// TwinCAT 3 PLC project ADSMotion
// ProgramVersion: 3.1.4024.0
// libraries:
//   Tc2_DataExchange, * (Beckhoff Automation GmbH)
//   Tc2_MC2, * (Beckhoff Automation GmbH)
//   Tc2_Standard, * (Beckhoff Automation GmbH)
//   Tc2_System, * (Beckhoff Automation GmbH)
//   Tc3_Module, * (Beckhoff Automation GmbH)
// project tree:
//   DUTs/ ST_variables.TcDUT
//   / PlcTask.TcTTO
//   POUs/ MAIN.TcPOU
// real-time tasks:
//   TASK PlcTask: cycle T#10ms, priority 20, ADS port 350
// motion (NC):
//   TASK NC-Task 1 SAF: cycle T#10ms, priority 4, ADS port 501
//   TASK NC-Task 1 SVB: cycle T#10ms, priority 8, ADS port 511
//   AXIS Axis 1 (id 1)
//     OtherSettings: AllowMotionCmdToSlave=true
//     encoder EncType=1
//     drive DrvType=5
//       Analog: TorqueSetpointScale=10, ScaleFactorActTorque=0.1
//       TimeComp: TaskDelayCycles=1
//     controller CtrType=1
//       CtrPara: PriorControlFactor=1
//         Observer: BandWidth=20

CONFIGURATION ADSMotion
    RESOURCE PLC ON TwinCAT3
        TASK PlcTask(INTERVAL := T#10ms, PRIORITY := 20);
        PROGRAM MAIN WITH PlcTask : MAIN;
    END_RESOURCE
END_CONFIGURATION

// ---- DUTs/ST_variables.TcDUT
TYPE ST_variables :
STRUCT
	bEnable   : BOOL;
    bStop     : BOOL;
    bMoveRel  : BOOL;
    rVelocity : REAL;
    rDistance : REAL;
END_STRUCT
END_TYPE

// ---- POUs/MAIN.TcPOU
PROGRAM MAIN
VAR
	//Write BOOL and REAL
	fbADSBoolEnable		: FB_WriteBoolOnDelta;
	fbADSBoolStop 		: FB_WriteBoolOnDelta;
	fbADSBoolRelMove 	: FB_WriteBoolOnDelta;
	fbADSRealVelocity	: FB_WriteRealOnDelta;
	fbADSRealDistance	: FB_WriteRealOnDelta;
	
    //ADS Comms Watchdoog
    fbWrWd : FB_WriteWatchdog;

		
	bEnabletx 		:BOOL; //Enable Controller
	bStoptx			: BOOL;
	bMoveReltx		: BOOL;
	rVelocitytx		: REAL;
	rDistancetx		: REAL;

	
END_VAR

fbWrWd(
    bEnable       := TRUE,
    sNetId        := '10.200.228.35.1.1',
    nPort         := 851,
    sVarName      := 'MAIN.nWatchdogRx',
    tWatchdogTime := T#1S
);

fbADSBoolEnable(
	bEnable:= TRUE , 
	sNetId:= '10.200.228.35.1.1', 
	nPort:= 851 , 
	sVarName:= 'MAIN.bEnable' , 
	bSignal:= bEnabletx , 
	tCycleTime:= T#1MS , 
	bSendNow:= FALSE );

fbADSBoolStop(
	bEnable:= TRUE , 
	sNetId:= '10.200.228.35.1.1', 
	nPort:= 851 , 
	sVarName:= 'MAIN.bStop' , 
	bSignal:= bStoptx , 
	tCycleTime:= T#1MS , 
	bSendNow:= FALSE );
	
fbADSBoolRelMove(
	bEnable:= TRUE , 
	sNetId:= '10.200.228.35.1.1', 
	nPort:= 851 , 
	sVarName:= 'MAIN.bMoveRel' , 
	bSignal:= bMoveReltx , 
	tCycleTime:= T#1MS , 
	bSendNow:= FALSE );
	
fbADSRealVelocity(
	bEnable:= TRUE, 
	sNetId:= '10.200.228.35.1.1' , 
	nPort:= 851 , 
	sVarName:= 'MAIN.rVelocity' , 
	fSignal:= rVelocitytx , 
	fLowerLimit:= 0.01 , 
	fUpperLimit:= 0.01 , 
	tCycleTime:= T#10MS, 
	bSendNow:= FALSE );
	
fbADSRealDistance(
	bEnable:= TRUE, 
	sNetId:= '10.200.228.35.1.1' , 
	nPort:= 851 , 
	sVarName:= 'MAIN.rDistance' , 
	fSignal:= rDistancetx , 
	fLowerLimit:= 0.01 , 
	fUpperLimit:= 0.01 , 
	tCycleTime:= T#10MS, 
	bSendNow:= FALSE );

END_PROGRAM
